FUNCTION_BLOCK FB_ServoMotor
VAR
    bEnable : BOOL;
END_VAR

END_FUNCTION_BLOCK

(* stored: POU FB_ServoMotor: Id {00000000-0000-0000-0000-000000000000} *)
